{attribute 'qualified_only'}
TYPE E_OBJECTS :
(
	UNDEFINED := 0,
	CYLINDER,
	DOOR,
	MOTOR
);
END_TYPE

(* stored: Version 1.1.0.1, ProductVersion 3.1.4024.12
   DUT E_OBJECTS: Id {6f2bf699-b7e9-4242-9deb-e129d6621c64} *)
